PROGRAM MAIN
VAR
END_VAR

END_PROGRAM

(* stored: Version 1.1.0.1
   POU MAIN: Id {d5ab113a-b34d-426c-8898-e61d97aa84f2} *)
